Omron Sysmac Studio project TROL_NX1P2_NS_Fev22 (Sysmac Studio 1.47.0.64008, StandardProject)

# Controller new_Controller_0: NX1P2-1140DT1 version 1.47
Units and slaves: Node1 : NX-ECC202 (E001); Unit 1 : NX-ID5442 (N5); Unit 2 : NX-ID5442 (N6); Unit 3 : NX-OD5256 (N7); Unit 4 : NX-OD5256 (N8); Unit 1 : NX-ID5142-1 (N1); Unit 2 : NX-ID5142-1 (N2); Unit 3 : NX-OD5256-1 (N3); Unit 4 : NX-OD5256-1 (N4)
Task PrimaryTask (priority 4, period or condition 2000): Program0

VAR_GLOBAL
    CH_CicloFarol : BOOL;  (* at BuiltInIO://cpu/#0/Input_Bit_00; published *)
    LMP_VM : BOOL;  (* at BuiltInIO://cpu/#0/Output_Bit_00; published *)
    LMP_VD : BOOL;  (* at BuiltInIO://cpu/#0/Output_Bit_01; published *)
    LMP_AM : BOOL;  (* at BuiltInIO://cpu/#0/Output_Bit_02; published *)
    Memo_Produto1 : ARRAY[0..9] OF LREAL;  (* published *)
    Memo_Produto2 : ARRAY[0..9] OF LREAL;  (* published *)
    Memo_Produção : ARRAY[0..9] OF LREAL;  (* published *)
    CH1_Produto1 : BOOL;  (* at ECAT://node#[1,1]/Input Bit 16 bits/Input Bit 00; published *)
    CH2_Produto2 : BOOL;  (* at ECAT://node#[1,1]/Input Bit 16 bits/Input Bit 01; published *)
    Alarmes : ARRAY[0..4] OF BOOL;  (* published *)
END_VAR

PROGRAM Program0
VAR
    TON_VM : TON;
    TMP_LMP_VM : TIME;
    TON_VD : TON;
    TMP_LMP_VD : TIME;
    TON_AM : TON;
    TMP_LMP_AM : TIME;
    Alm1 : ARRAY[0..4] OF BOOL;
END_VAR
VAR_EXTERNAL
    CH_CicloFarol : BOOL;
    LMP_VM : BOOL;
    LMP_VD : BOOL;
    LMP_AM : BOOL;
    CH2_Produto2 : BOOL;
    CH1_Produto1 : BOOL;
    Memo_Produção : ARRAY[0..9] OF LREAL;
    Memo_Produto1 : ARRAY[0..9] OF LREAL;
    Memo_Produto2 : ARRAY[0..9] OF LREAL;
    Alarmes : ARRAY[0..4] OF BOOL;
END_VAR

(* Section Semáforo: ladder, written here as Structured Text *)

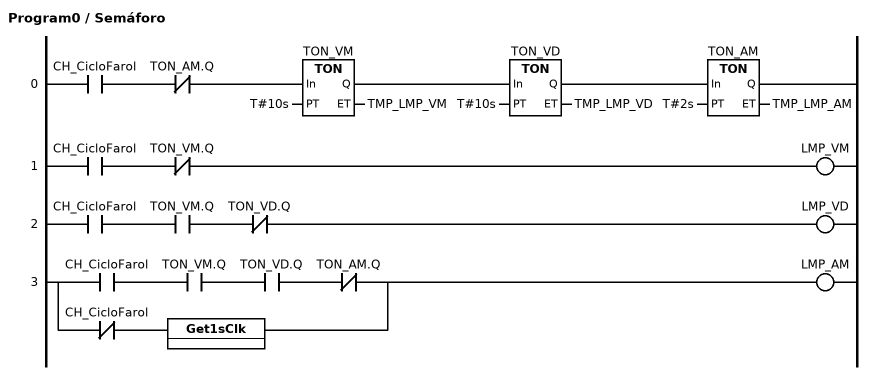
(* Rung 0 *)
TON_VM(In := CH_CicloFarol AND NOT TON_AM.Q, PT := T#10s, ET => TMP_LMP_VM);
TON_VD(In := TON_VM.Q, PT := T#10s, ET => TMP_LMP_VD);
TON_AM(In := TON_VD.Q, PT := T#2s, ET => TMP_LMP_AM);
(* Rung 1 *)
LMP_VM := CH_CicloFarol AND NOT TON_VM.Q;
(* Rung 2 *)
LMP_VD := CH_CicloFarol AND TON_VM.Q AND NOT TON_VD.Q;
(* Rung 3 *)
LMP_AM := (CH_CicloFarol AND TON_VM.Q AND TON_VD.Q AND NOT TON_AM.Q) OR (NOT CH_CicloFarol AND Get1sClk());

(* Section Receita: ladder, written here as Structured Text *)

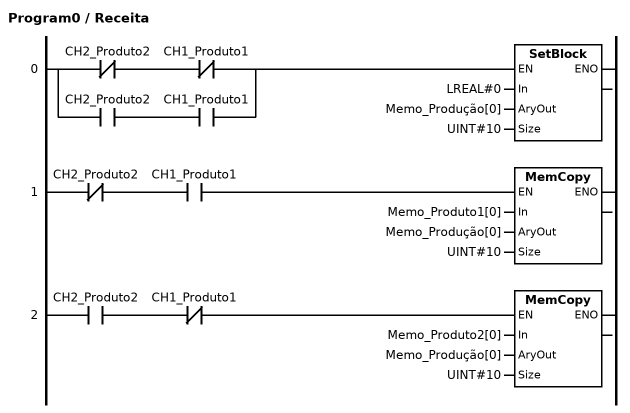
(* Rung 0 *)
IF (NOT CH2_Produto2 AND NOT CH1_Produto1) OR (CH2_Produto2 AND CH1_Produto1) THEN
    SetBlock(In := LREAL#0, AryOut := Memo_Produção[0], Size := UINT#10);
END_IF;
(* Rung 1 *)
IF NOT CH2_Produto2 AND CH1_Produto1 THEN
    MemCopy(In := Memo_Produto1[0], AryOut := Memo_Produção[0], Size := UINT#10);
END_IF;
(* Rung 2 *)
IF CH2_Produto2 AND NOT CH1_Produto1 THEN
    MemCopy(In := Memo_Produto2[0], AryOut := Memo_Produção[0], Size := UINT#10);
END_IF;

(* Section Alarmas: ladder, written here as Structured Text *)

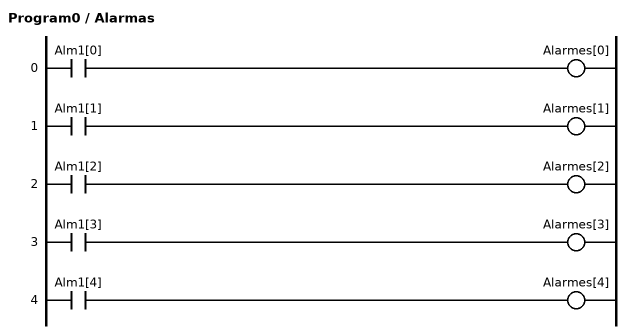
(* Rung 0 *)
Alarmes[0] := Alm1[0];
(* Rung 1 *)
Alarmes[1] := Alm1[1];
(* Rung 2 *)
Alarmes[2] := Alm1[2];
(* Rung 3 *)
Alarmes[3] := Alm1[3];
(* Rung 4 *)
Alarmes[4] := Alm1[4];
END_PROGRAM